// TIA Portal project "lab2" (V15.1)

(* hardware
DEVICE "S71500/ET200MP station_1"  S7-1500 station
   slot 0: "Rail_0"  Rack  6ES7 590-1***0-0AA0
   slot 1: "PLC_1"  CPU 1512C-1 PN  6ES7 512-1CK01-0AB0  V2.6
      slot 3: "CPU display_1"  6ES7591-1AA00-0AA0
*)

// ===== PLC "PLC_1"  CPU 1512C-1 PN =====

VAR_GLOBAL   // PLC tag table "Default tag table"
   "DIGITALNI_ULAZ_KLIP_1_LEVO_NO" AT %I10.6 : Bool;
   "DIGITALNI_ULAZ_KLIP_1_DESNO_NO" AT %I10.7 : Bool;
   "DIGITALNI_ULAZ_KLIP_2_LEVO_NO" AT %I10.4 : Bool;
   "DIGITALNI_ULAZ_KLIP_2_DESNO_NO" AT %I10.5 : Bool;
   "DIGITALNI_ULAZ_KLIP_3_LEVO_NO" AT %I10.2 : Bool;
   "DIGITALNI_ULAZ_KLIP_3_DESNO_NO" AT %I10.3 : Bool;
   "DIGITALNI_ULAZ_KLIP_4_LEVO_NO" AT %I10.0 : Bool;
   "DIGITALNI_ULAZ_KLIP_4_DESNO_NO" AT %I10.1 : Bool;
   "DIGITALNI_IZLAZ_KLIP_1_DESNO" AT %Q4.5 : Bool;
   "DIGITALNI_IZLAZ_KLIP_2_DESNO" AT %Q4.4 : Bool;
   "DIGITALNI_IZLAZ_KLIP_3_LEVO" AT %Q4.3 : Bool;
   "DIGITALNI_IZLAZ_KLIP_3_DESNO" AT %Q4.2 : Bool;
   "DIGITALNI_IZLAZ_KLIP_4_LEVO" AT %Q4.1 : Bool;
   "DIGITALNI_IZLAZ_KLIP_4_DESNO" AT %Q4.0 : Bool;
   "ANALOGNI_ULAZ_POZICIJA_KLIP_1" AT %IW0 : Word;
END_VAR

DATA_BLOCK "DB"   // DB1
{ S7_Optimized_Access := 'TRUE' }
VERSION : 0.1
   VAR
      TRENUTNO_STANJE : Int := 0;
      "POZICIJA_KLIP_1_50%" : Int := 3638;
      "POZICIJA_KLIP_1_60%" : Int := 4046;
      "POZICIJA_KLIP_1_70%" : Int := 4453;
      KLIPOVI_RESETOVANI : Bool;
   END_VAR
BEGIN
END_DATA_BLOCK

// folder: System blocks/Program resources

DATA_BLOCK "KORAK_2_TAJMER"   // DB2
{ S7_Optimized_Access := 'TRUE' }
AUTHOR : Simatic
FAMILY : IEC
NAME : IEC_TMR
VERSION : 1.0
// stored: InstanceOfName IEC_TIMER
"IEC_TIMER"
BEGIN
END_DATA_BLOCK

DATA_BLOCK "RESETOVANJE_KLIPOVA_TAJMER"   // DB3
{ S7_Optimized_Access := 'TRUE' }
AUTHOR : Simatic
FAMILY : IEC
NAME : IEC_TMR
VERSION : 1.0
// stored: InstanceOfName IEC_TIMER
"IEC_TIMER"
BEGIN
END_DATA_BLOCK

DATA_BLOCK "KORAK_4_BROJAC_ITERACIJA"   // DB4
{ S7_Optimized_Access := 'TRUE' }
AUTHOR : Simatic
FAMILY : IEC
NAME : CNTR
VERSION : 1.0
// stored: InstanceOfName IEC_COUNTER
"IEC_COUNTER"
BEGIN
END_DATA_BLOCK

// folder: (top level)

FUNCTION "OBRADA_KORAK_0" : Void   // FC1, LAD
{ S7_Optimized_Access := 'TRUE' }
VERSION : 0.1
BEGIN

REGION Network 1
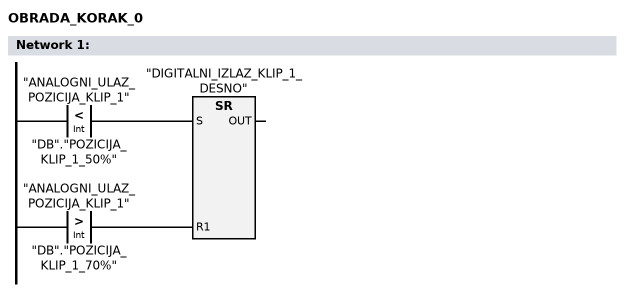
   RUNG wire#powerrail
      { S7_Templates := "SrcType := Int" } LT_Contact(in1 := "ANALOGNI_ULAZ_POZICIJA_KLIP_1", in2 := "DB"."POZICIJA_KLIP_1_50%")
      S_SR(operand := "DIGITALNI_IZLAZ_KLIP_1_DESNO", r1 := wire#w1)
   END_RUNG
   RUNG wire#powerrail
      { S7_Templates := "SrcType := Int" } GT_Contact(in1 := "ANALOGNI_ULAZ_POZICIJA_KLIP_1", in2 := "DB"."POZICIJA_KLIP_1_70%")
   END_RUNG wire#w1
   // the same network as SCL:
   IF "ANALOGNI_ULAZ_POZICIJA_KLIP_1" < "DB"."POZICIJA_KLIP_1_50%" THEN
       "DIGITALNI_IZLAZ_KLIP_1_DESNO" := TRUE;   // SR flip-flop
   END_IF;
   IF "ANALOGNI_ULAZ_POZICIJA_KLIP_1" > "DB"."POZICIJA_KLIP_1_70%" THEN
       "DIGITALNI_IZLAZ_KLIP_1_DESNO" := FALSE;
   END_IF;
END_REGION
END_FUNCTION

FUNCTION "PRELAZ_KORAK_0_U_KORAK_1" : Void   // FC2, LAD
{ S7_Optimized_Access := 'TRUE' }
VERSION : 0.1
BEGIN

REGION Network 1
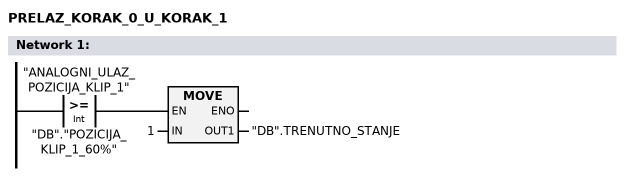
   RUNG wire#powerrail
      { S7_Templates := "SrcType := Int" } GE_Contact(in1 := "ANALOGNI_ULAZ_POZICIJA_KLIP_1", in2 := "DB"."POZICIJA_KLIP_1_60%")
      Move(in := 1, out1 => "DB".TRENUTNO_STANJE)
   END_RUNG
   // the same network as SCL:
   IF "ANALOGNI_ULAZ_POZICIJA_KLIP_1" >= "DB"."POZICIJA_KLIP_1_60%" THEN "DB".TRENUTNO_STANJE := 1; END_IF;
END_REGION
END_FUNCTION

FUNCTION "OBRADA_KORAK_1" : Void   // FC3, LAD
{ S7_Optimized_Access := 'TRUE' }
VERSION : 0.1
BEGIN

REGION Network 1
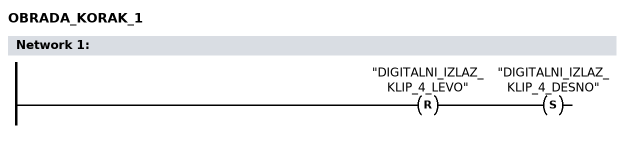
   RUNG wire#powerrail
      R_Coil( "DIGITALNI_IZLAZ_KLIP_4_LEVO" )
      S_Coil( "DIGITALNI_IZLAZ_KLIP_4_DESNO" )
   END_RUNG
   // the same network as SCL:
   "DIGITALNI_IZLAZ_KLIP_4_LEVO" := FALSE;
   "DIGITALNI_IZLAZ_KLIP_4_DESNO" := TRUE;
END_REGION
END_FUNCTION

FUNCTION "PRELAZ_KORAK_1_U_KORAK_2" : Void   // FC4, LAD
{ S7_Optimized_Access := 'TRUE' }
VERSION : 0.1
BEGIN

REGION Network 1
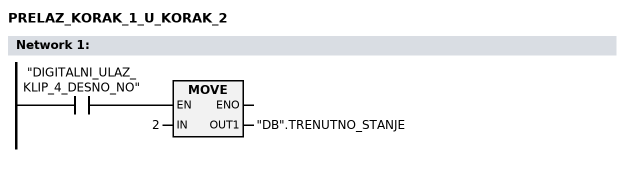
   RUNG wire#powerrail
      Contact( "DIGITALNI_ULAZ_KLIP_4_DESNO_NO" )
      Move(in := 2, out1 => "DB".TRENUTNO_STANJE)
   END_RUNG
   // the same network as SCL:
   IF "DIGITALNI_ULAZ_KLIP_4_DESNO_NO" THEN "DB".TRENUTNO_STANJE := 2; END_IF;
END_REGION
END_FUNCTION

FUNCTION "IZVRSENJE_SEKVENCE" : Void   // FC5, LAD
{ S7_Optimized_Access := 'TRUE' }
VERSION : 0.1
BEGIN

REGION Network 1
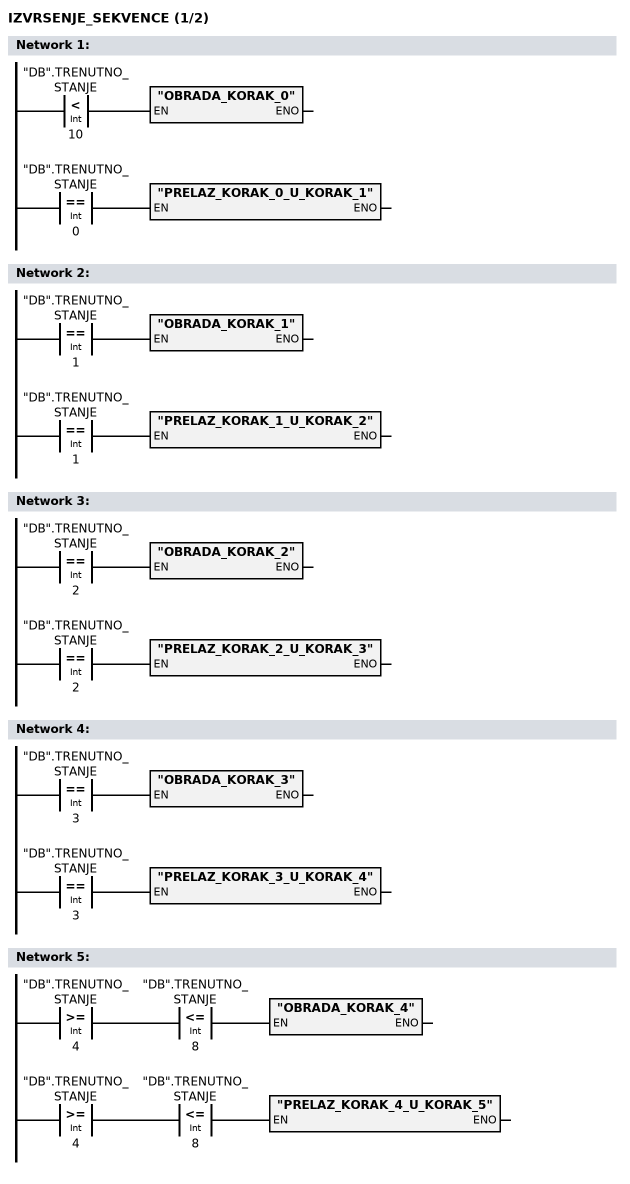
   RUNG wire#powerrail
      { S7_Templates := "SrcType := Int" } LT_Contact(in1 := "DB".TRENUTNO_STANJE, in2 := 10)
      "OBRADA_KORAK_0"()
   END_RUNG
   RUNG wire#powerrail
      { S7_Templates := "SrcType := Int" } EQ_Contact(in1 := "DB".TRENUTNO_STANJE, in2 := 0)
      "PRELAZ_KORAK_0_U_KORAK_1"()
   END_RUNG
   // the same network as SCL:
   IF "DB".TRENUTNO_STANJE < 10 THEN "OBRADA_KORAK_0"(); END_IF;
   IF "DB".TRENUTNO_STANJE = 0 THEN "PRELAZ_KORAK_0_U_KORAK_1"(); END_IF;
END_REGION

REGION Network 2
   RUNG wire#powerrail
      { S7_Templates := "SrcType := Int" } EQ_Contact(in1 := "DB".TRENUTNO_STANJE, in2 := 1)
      "OBRADA_KORAK_1"()
   END_RUNG
   RUNG wire#powerrail
      { S7_Templates := "SrcType := Int" } EQ_Contact(in1 := "DB".TRENUTNO_STANJE, in2 := 1)
      "PRELAZ_KORAK_1_U_KORAK_2"()
   END_RUNG
   // the same network as SCL:
   IF "DB".TRENUTNO_STANJE = 1 THEN "OBRADA_KORAK_1"(); END_IF;
   IF "DB".TRENUTNO_STANJE = 1 THEN "PRELAZ_KORAK_1_U_KORAK_2"(); END_IF;
END_REGION

REGION Network 3
   RUNG wire#powerrail
      { S7_Templates := "SrcType := Int" } EQ_Contact(in1 := "DB".TRENUTNO_STANJE, in2 := 2)
      "OBRADA_KORAK_2"()
   END_RUNG
   RUNG wire#powerrail
      { S7_Templates := "SrcType := Int" } EQ_Contact(in1 := "DB".TRENUTNO_STANJE, in2 := 2)
      "PRELAZ_KORAK_2_U_KORAK_3"()
   END_RUNG
   // the same network as SCL:
   IF "DB".TRENUTNO_STANJE = 2 THEN "OBRADA_KORAK_2"(); END_IF;
   IF "DB".TRENUTNO_STANJE = 2 THEN "PRELAZ_KORAK_2_U_KORAK_3"(); END_IF;
END_REGION

REGION Network 4
   RUNG wire#powerrail
      { S7_Templates := "SrcType := Int" } EQ_Contact(in1 := "DB".TRENUTNO_STANJE, in2 := 3)
      "OBRADA_KORAK_3"()
   END_RUNG
   RUNG wire#powerrail
      { S7_Templates := "SrcType := Int" } EQ_Contact(in1 := "DB".TRENUTNO_STANJE, in2 := 3)
      "PRELAZ_KORAK_3_U_KORAK_4"()
   END_RUNG
   // the same network as SCL:
   IF "DB".TRENUTNO_STANJE = 3 THEN "OBRADA_KORAK_3"(); END_IF;
   IF "DB".TRENUTNO_STANJE = 3 THEN "PRELAZ_KORAK_3_U_KORAK_4"(); END_IF;
END_REGION

REGION Network 5
   RUNG wire#powerrail
      { S7_Templates := "SrcType := Int" } GE_Contact(in1 := "DB".TRENUTNO_STANJE, in2 := 4)
      { S7_Templates := "SrcType := Int" } LE_Contact(in1 := "DB".TRENUTNO_STANJE, in2 := 8)
      "OBRADA_KORAK_4"()
   END_RUNG
   RUNG wire#powerrail
      { S7_Templates := "SrcType := Int" } GE_Contact(in1 := "DB".TRENUTNO_STANJE, in2 := 4)
      { S7_Templates := "SrcType := Int" } LE_Contact(in1 := "DB".TRENUTNO_STANJE, in2 := 8)
      "PRELAZ_KORAK_4_U_KORAK_5"()
   END_RUNG
   // the same network as SCL:
   IF ("DB".TRENUTNO_STANJE >= 4) AND ("DB".TRENUTNO_STANJE <= 8) THEN "OBRADA_KORAK_4"(); END_IF;
   IF ("DB".TRENUTNO_STANJE >= 4) AND ("DB".TRENUTNO_STANJE <= 8) THEN "PRELAZ_KORAK_4_U_KORAK_5"(); END_IF;
END_REGION

REGION Network 6
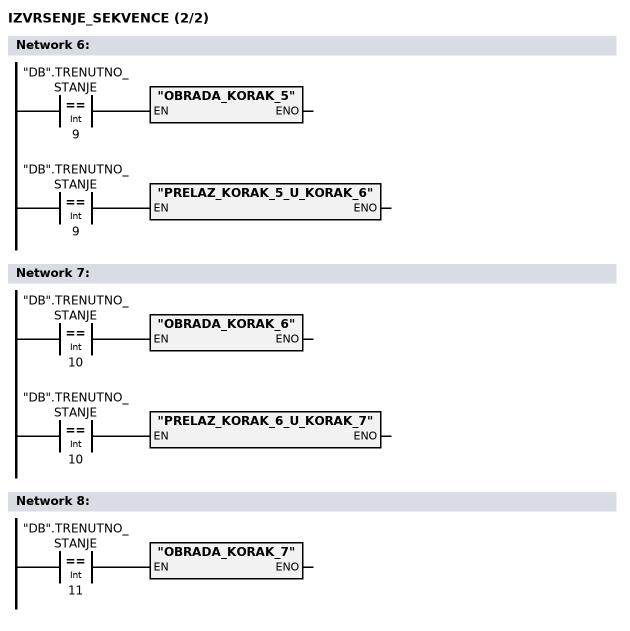
   RUNG wire#powerrail
      { S7_Templates := "SrcType := Int" } EQ_Contact(in1 := "DB".TRENUTNO_STANJE, in2 := 9)
      "OBRADA_KORAK_5"()
   END_RUNG
   RUNG wire#powerrail
      { S7_Templates := "SrcType := Int" } EQ_Contact(in1 := "DB".TRENUTNO_STANJE, in2 := 9)
      "PRELAZ_KORAK_5_U_KORAK_6"()
   END_RUNG
   // the same network as SCL:
   IF "DB".TRENUTNO_STANJE = 9 THEN "OBRADA_KORAK_5"(); END_IF;
   IF "DB".TRENUTNO_STANJE = 9 THEN "PRELAZ_KORAK_5_U_KORAK_6"(); END_IF;
END_REGION

REGION Network 7
   RUNG wire#powerrail
      { S7_Templates := "SrcType := Int" } EQ_Contact(in1 := "DB".TRENUTNO_STANJE, in2 := 10)
      "OBRADA_KORAK_6"()
   END_RUNG
   RUNG wire#powerrail
      { S7_Templates := "SrcType := Int" } EQ_Contact(in1 := "DB".TRENUTNO_STANJE, in2 := 10)
      "PRELAZ_KORAK_6_U_KORAK_7"()
   END_RUNG
   // the same network as SCL:
   IF "DB".TRENUTNO_STANJE = 10 THEN "OBRADA_KORAK_6"(); END_IF;
   IF "DB".TRENUTNO_STANJE = 10 THEN "PRELAZ_KORAK_6_U_KORAK_7"(); END_IF;
END_REGION

REGION Network 8
   RUNG wire#powerrail
      { S7_Templates := "SrcType := Int" } EQ_Contact(in1 := "DB".TRENUTNO_STANJE, in2 := 11)
      "OBRADA_KORAK_7"()
   END_RUNG
   // the same network as SCL:
   IF "DB".TRENUTNO_STANJE = 11 THEN "OBRADA_KORAK_7"(); END_IF;
END_REGION
END_FUNCTION

FUNCTION "OBRADA_KORAK_2" : Void   // FC6, LAD
{ S7_Optimized_Access := 'TRUE' }
VERSION : 0.1
   VAR CONSTANT
      TRUE_CONSTANT : Bool := true;
   END_VAR
BEGIN

REGION Network 1
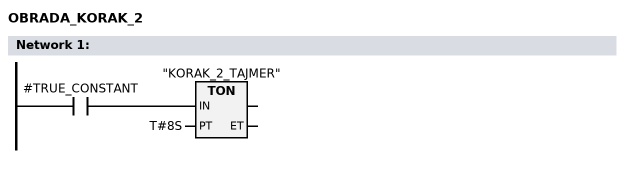
   "KORAK_2_TAJMER".TON(IN := #TRUE_CONSTANT, PT := T#8S);
END_REGION
END_FUNCTION

FUNCTION "PRELAZ_KORAK_2_U_KORAK_3" : Void   // FC7, LAD
{ S7_Optimized_Access := 'TRUE' }
VERSION : 0.1
BEGIN

REGION Network 1
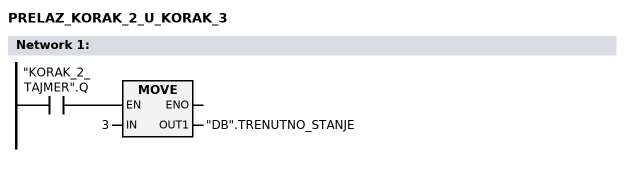
   RUNG wire#powerrail
      Contact( "KORAK_2_TAJMER".Q )
      Move(in := 3, out1 => "DB".TRENUTNO_STANJE)
   END_RUNG
   // the same network as SCL:
   IF "KORAK_2_TAJMER".Q THEN "DB".TRENUTNO_STANJE := 3; END_IF;
END_REGION
END_FUNCTION

FUNCTION "OBRADA_KORAK_3" : Void   // FC8, LAD
{ S7_Optimized_Access := 'TRUE' }
VERSION : 0.1
BEGIN

REGION Network 1
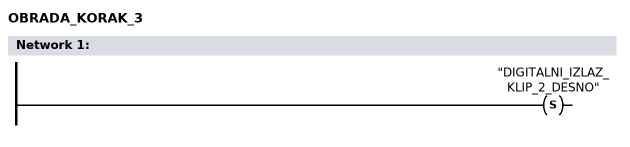
   RUNG wire#powerrail
      S_Coil( "DIGITALNI_IZLAZ_KLIP_2_DESNO" )
   END_RUNG
   // the same network as SCL:
   "DIGITALNI_IZLAZ_KLIP_2_DESNO" := TRUE;
END_REGION
END_FUNCTION

FUNCTION "PRELAZ_KORAK_3_U_KORAK_4" : Void   // FC9, LAD
{ S7_Optimized_Access := 'TRUE' }
VERSION : 0.1
BEGIN

REGION Network 1
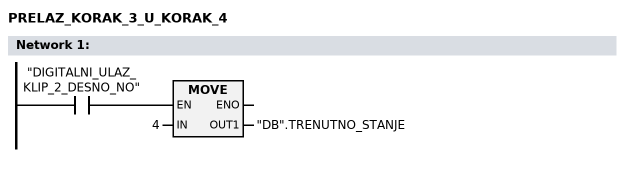
   RUNG wire#powerrail
      Contact( "DIGITALNI_ULAZ_KLIP_2_DESNO_NO" )
      Move(in := 4, out1 => "DB".TRENUTNO_STANJE)
   END_RUNG
   // the same network as SCL:
   IF "DIGITALNI_ULAZ_KLIP_2_DESNO_NO" THEN "DB".TRENUTNO_STANJE := 4; END_IF;
END_REGION
END_FUNCTION

FUNCTION "OBRADA_KORAK_4" : Void   // FC10, LAD
{ S7_Optimized_Access := 'TRUE' }
VERSION : 0.1
BEGIN

REGION Network 1
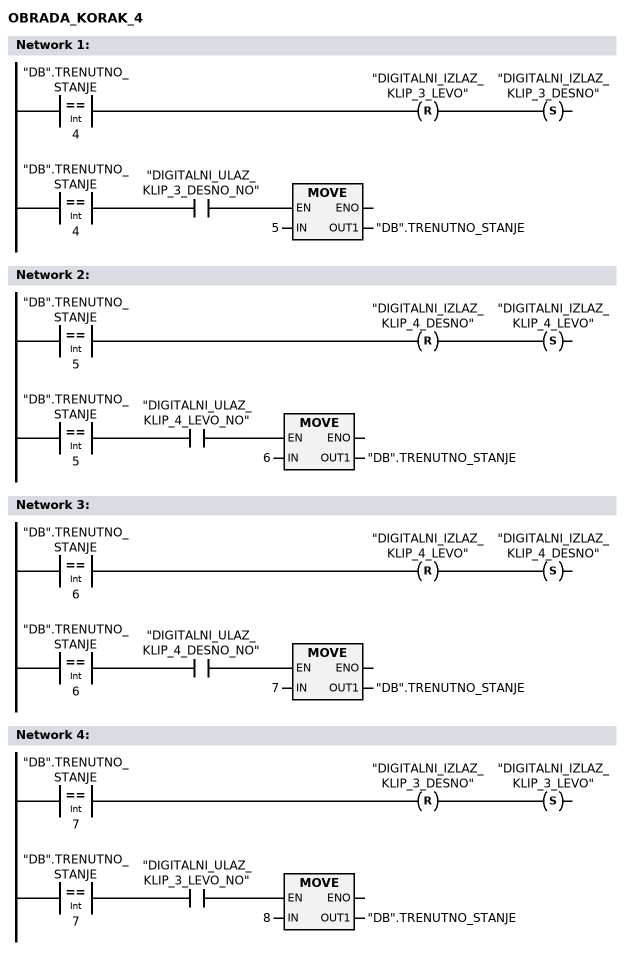
   RUNG wire#powerrail
      { S7_Templates := "SrcType := Int" } EQ_Contact(in1 := "DB".TRENUTNO_STANJE, in2 := 4)
      R_Coil( "DIGITALNI_IZLAZ_KLIP_3_LEVO" )
      S_Coil( "DIGITALNI_IZLAZ_KLIP_3_DESNO" )
   END_RUNG
   RUNG wire#powerrail
      { S7_Templates := "SrcType := Int" } EQ_Contact(in1 := "DB".TRENUTNO_STANJE, in2 := 4)
      Contact( "DIGITALNI_ULAZ_KLIP_3_DESNO_NO" )
      Move(in := 5, out1 => "DB".TRENUTNO_STANJE)
   END_RUNG
   // the same network as SCL:
   IF "DB".TRENUTNO_STANJE = 4 THEN
       "DIGITALNI_IZLAZ_KLIP_3_LEVO" := FALSE;
       "DIGITALNI_IZLAZ_KLIP_3_DESNO" := TRUE;
   END_IF;
   IF ("DB".TRENUTNO_STANJE = 4) AND "DIGITALNI_ULAZ_KLIP_3_DESNO_NO" THEN "DB".TRENUTNO_STANJE := 5; END_IF;
END_REGION

REGION Network 2
   RUNG wire#powerrail
      { S7_Templates := "SrcType := Int" } EQ_Contact(in1 := "DB".TRENUTNO_STANJE, in2 := 5)
      R_Coil( "DIGITALNI_IZLAZ_KLIP_4_DESNO" )
      S_Coil( "DIGITALNI_IZLAZ_KLIP_4_LEVO" )
   END_RUNG
   RUNG wire#powerrail
      { S7_Templates := "SrcType := Int" } EQ_Contact(in1 := "DB".TRENUTNO_STANJE, in2 := 5)
      Contact( "DIGITALNI_ULAZ_KLIP_4_LEVO_NO" )
      Move(in := 6, out1 => "DB".TRENUTNO_STANJE)
   END_RUNG
   // the same network as SCL:
   IF "DB".TRENUTNO_STANJE = 5 THEN
       "DIGITALNI_IZLAZ_KLIP_4_DESNO" := FALSE;
       "DIGITALNI_IZLAZ_KLIP_4_LEVO" := TRUE;
   END_IF;
   IF ("DB".TRENUTNO_STANJE = 5) AND "DIGITALNI_ULAZ_KLIP_4_LEVO_NO" THEN "DB".TRENUTNO_STANJE := 6; END_IF;
END_REGION

REGION Network 3
   RUNG wire#powerrail
      { S7_Templates := "SrcType := Int" } EQ_Contact(in1 := "DB".TRENUTNO_STANJE, in2 := 6)
      R_Coil( "DIGITALNI_IZLAZ_KLIP_4_LEVO" )
      S_Coil( "DIGITALNI_IZLAZ_KLIP_4_DESNO" )
   END_RUNG
   RUNG wire#powerrail
      { S7_Templates := "SrcType := Int" } EQ_Contact(in1 := "DB".TRENUTNO_STANJE, in2 := 6)
      Contact( "DIGITALNI_ULAZ_KLIP_4_DESNO_NO" )
      Move(in := 7, out1 => "DB".TRENUTNO_STANJE)
   END_RUNG
   // the same network as SCL:
   IF "DB".TRENUTNO_STANJE = 6 THEN
       "DIGITALNI_IZLAZ_KLIP_4_LEVO" := FALSE;
       "DIGITALNI_IZLAZ_KLIP_4_DESNO" := TRUE;
   END_IF;
   IF ("DB".TRENUTNO_STANJE = 6) AND "DIGITALNI_ULAZ_KLIP_4_DESNO_NO" THEN "DB".TRENUTNO_STANJE := 7; END_IF;
END_REGION

REGION Network 4
   RUNG wire#powerrail
      { S7_Templates := "SrcType := Int" } EQ_Contact(in1 := "DB".TRENUTNO_STANJE, in2 := 7)
      R_Coil( "DIGITALNI_IZLAZ_KLIP_3_DESNO" )
      S_Coil( "DIGITALNI_IZLAZ_KLIP_3_LEVO" )
   END_RUNG
   RUNG wire#powerrail
      { S7_Templates := "SrcType := Int" } EQ_Contact(in1 := "DB".TRENUTNO_STANJE, in2 := 7)
      Contact( "DIGITALNI_ULAZ_KLIP_3_LEVO_NO" )
      Move(in := 8, out1 => "DB".TRENUTNO_STANJE)
   END_RUNG
   // the same network as SCL:
   IF "DB".TRENUTNO_STANJE = 7 THEN
       "DIGITALNI_IZLAZ_KLIP_3_DESNO" := FALSE;
       "DIGITALNI_IZLAZ_KLIP_3_LEVO" := TRUE;
   END_IF;
   IF ("DB".TRENUTNO_STANJE = 7) AND "DIGITALNI_ULAZ_KLIP_3_LEVO_NO" THEN "DB".TRENUTNO_STANJE := 8; END_IF;
END_REGION
END_FUNCTION

FUNCTION "PRELAZ_KORAK_4_U_KORAK_5" : Void   // FC11, LAD
{ S7_Optimized_Access := 'TRUE' }
VERSION : 0.1
BEGIN

REGION Network 1
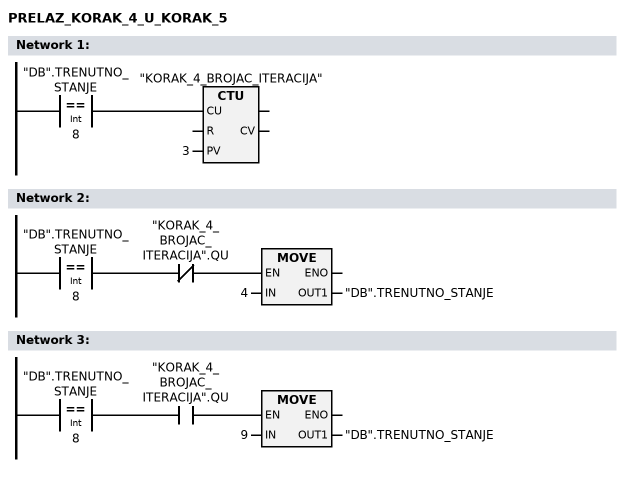
   "KORAK_4_BROJAC_ITERACIJA".CTU(CU := "DB".TRENUTNO_STANJE = 8, PV := 3);
END_REGION

REGION Network 2
   RUNG wire#powerrail
      { S7_Templates := "SrcType := Int" } EQ_Contact(in1 := "DB".TRENUTNO_STANJE, in2 := 8)
      I_Contact( "KORAK_4_BROJAC_ITERACIJA".QU )
      Move(in := 4, out1 => "DB".TRENUTNO_STANJE)
   END_RUNG
   // the same network as SCL:
   IF ("DB".TRENUTNO_STANJE = 8) AND NOT "KORAK_4_BROJAC_ITERACIJA".QU THEN
       "DB".TRENUTNO_STANJE := 4;
   END_IF;
END_REGION

REGION Network 3
   RUNG wire#powerrail
      { S7_Templates := "SrcType := Int" } EQ_Contact(in1 := "DB".TRENUTNO_STANJE, in2 := 8)
      Contact( "KORAK_4_BROJAC_ITERACIJA".QU )
      Move(in := 9, out1 => "DB".TRENUTNO_STANJE)
   END_RUNG
   // the same network as SCL:
   IF ("DB".TRENUTNO_STANJE = 8) AND "KORAK_4_BROJAC_ITERACIJA".QU THEN "DB".TRENUTNO_STANJE := 9; END_IF;
END_REGION
END_FUNCTION

FUNCTION "OBRADA_KORAK_5" : Void   // FC12, LAD
{ S7_Optimized_Access := 'TRUE' }
VERSION : 0.1
BEGIN

REGION Network 1
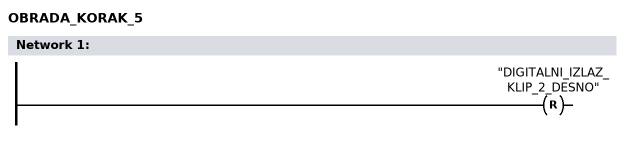
   RUNG wire#powerrail
      R_Coil( "DIGITALNI_IZLAZ_KLIP_2_DESNO" )
   END_RUNG
   // the same network as SCL:
   "DIGITALNI_IZLAZ_KLIP_2_DESNO" := FALSE;
END_REGION
END_FUNCTION

FUNCTION "PRELAZ_KORAK_5_U_KORAK_6" : Void   // FC13, LAD
{ S7_Optimized_Access := 'TRUE' }
VERSION : 0.1
BEGIN

REGION Network 1
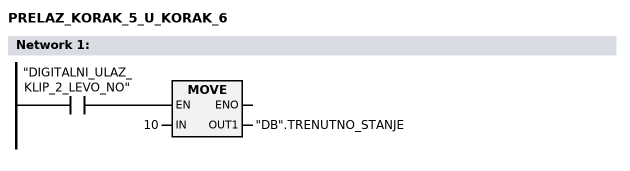
   RUNG wire#powerrail
      Contact( "DIGITALNI_ULAZ_KLIP_2_LEVO_NO" )
      Move(in := 10, out1 => "DB".TRENUTNO_STANJE)
   END_RUNG
   // the same network as SCL:
   IF "DIGITALNI_ULAZ_KLIP_2_LEVO_NO" THEN "DB".TRENUTNO_STANJE := 10; END_IF;
END_REGION
END_FUNCTION

FUNCTION "OBRADA_KORAK_6" : Void   // FC14, LAD
{ S7_Optimized_Access := 'TRUE' }
VERSION : 0.1
BEGIN

REGION Network 1
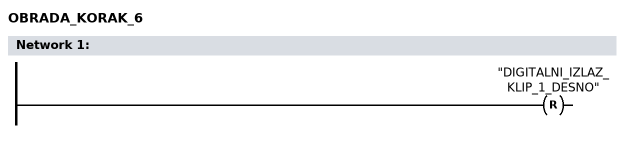
   RUNG wire#powerrail
      R_Coil( "DIGITALNI_IZLAZ_KLIP_1_DESNO" )
   END_RUNG
   // the same network as SCL:
   "DIGITALNI_IZLAZ_KLIP_1_DESNO" := FALSE;
END_REGION
END_FUNCTION

FUNCTION "PRELAZ_KORAK_6_U_KORAK_7" : Void   // FC15, LAD
{ S7_Optimized_Access := 'TRUE' }
VERSION : 0.1
BEGIN

REGION Network 1
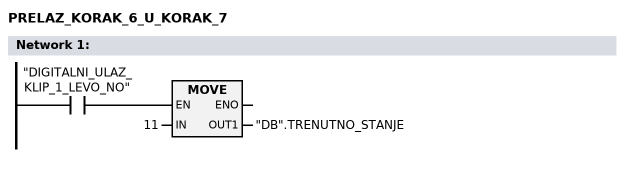
   RUNG wire#powerrail
      Contact( "DIGITALNI_ULAZ_KLIP_1_LEVO_NO" )
      Move(in := 11, out1 => "DB".TRENUTNO_STANJE)
   END_RUNG
   // the same network as SCL:
   IF "DIGITALNI_ULAZ_KLIP_1_LEVO_NO" THEN "DB".TRENUTNO_STANJE := 11; END_IF;
END_REGION
END_FUNCTION

FUNCTION "OBRADA_KORAK_7" : Void   // FC16, LAD
{ S7_Optimized_Access := 'TRUE' }
VERSION : 0.1
BEGIN

REGION Network 1
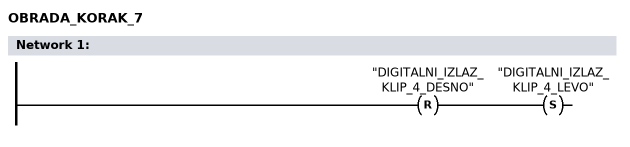
   RUNG wire#powerrail
      R_Coil( "DIGITALNI_IZLAZ_KLIP_4_DESNO" )
      S_Coil( "DIGITALNI_IZLAZ_KLIP_4_LEVO" )
   END_RUNG
   // the same network as SCL:
   "DIGITALNI_IZLAZ_KLIP_4_DESNO" := FALSE;
   "DIGITALNI_IZLAZ_KLIP_4_LEVO" := TRUE;
END_REGION
END_FUNCTION

ORGANIZATION_BLOCK "Main"   // OB1, LAD, ProgramCycle
TITLE = "Main Program Sweep (Cycle)"
{ S7_Optimized_Access := 'TRUE' }
VERSION : 0.1
   VAR_INPUT
      Initial_Call : Bool;   // Initial call of this OB
      Remanence : Bool;   // =True, if remanent data are available
   END_VAR
BEGIN

REGION Network 1
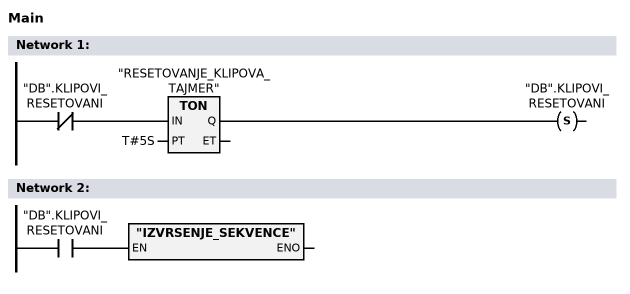
   "RESETOVANJE_KLIPOVA_TAJMER".TON(IN := NOT "DB".KLIPOVI_RESETOVANI, PT := T#5S);
   IF "RESETOVANJE_KLIPOVA_TAJMER".Q THEN "DB".KLIPOVI_RESETOVANI := TRUE; END_IF;
END_REGION

REGION Network 2
   RUNG wire#powerrail
      Contact( "DB".KLIPOVI_RESETOVANI )
      "IZVRSENJE_SEKVENCE"()
   END_RUNG
   // the same network as SCL:
   IF "DB".KLIPOVI_RESETOVANI THEN "IZVRSENJE_SEKVENCE"(); END_IF;
END_REGION
END_ORGANIZATION_BLOCK

ORGANIZATION_BLOCK "Startup"   // OB100, LAD, Startup
TITLE = "Complete Restart"
{ S7_Optimized_Access := 'TRUE' }
VERSION : 0.1
   VAR_INPUT
      LostRetentive : Bool;   // True if retentive data are lost
      LostRTC : Bool;   // True if date and time are lost
   END_VAR
BEGIN

REGION Network 1
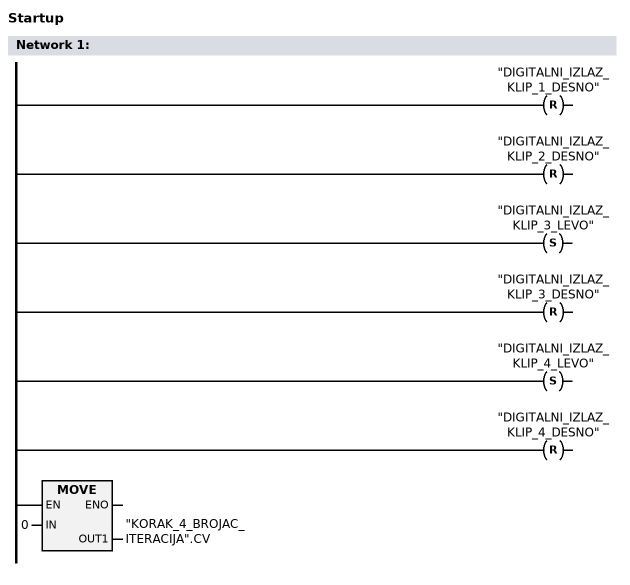
   RUNG wire#powerrail
      R_Coil( "DIGITALNI_IZLAZ_KLIP_1_DESNO" )
   END_RUNG
   RUNG wire#powerrail
      R_Coil( "DIGITALNI_IZLAZ_KLIP_2_DESNO" )
   END_RUNG
   RUNG wire#powerrail
      S_Coil( "DIGITALNI_IZLAZ_KLIP_3_LEVO" )
   END_RUNG
   RUNG wire#powerrail
      R_Coil( "DIGITALNI_IZLAZ_KLIP_3_DESNO" )
   END_RUNG
   RUNG wire#powerrail
      S_Coil( "DIGITALNI_IZLAZ_KLIP_4_LEVO" )
   END_RUNG
   RUNG wire#powerrail
      R_Coil( "DIGITALNI_IZLAZ_KLIP_4_DESNO" )
   END_RUNG
   RUNG wire#powerrail
      Move(in := 0, out1 => "KORAK_4_BROJAC_ITERACIJA".CV)
   END_RUNG
   // the same network as SCL:
   "DIGITALNI_IZLAZ_KLIP_1_DESNO" := FALSE;
   "DIGITALNI_IZLAZ_KLIP_2_DESNO" := FALSE;
   "DIGITALNI_IZLAZ_KLIP_3_LEVO" := TRUE;
   "DIGITALNI_IZLAZ_KLIP_3_DESNO" := FALSE;
   "DIGITALNI_IZLAZ_KLIP_4_LEVO" := TRUE;
   "DIGITALNI_IZLAZ_KLIP_4_DESNO" := FALSE;
   "KORAK_4_BROJAC_ITERACIJA".CV := 0;
END_REGION
END_ORGANIZATION_BLOCK